FUNCTION_BLOCK FB_MqttBlindInputAdapter IMPLEMENTS I_CyclicExecution, I_MqttMessageReceiver, I_MqttDeviceDiscoveryProvider
VAR_INPUT
	POS : BYTE;	// Feedback of blind position
END_VAR
VAR_OUTPUT
	Q : BOOL;  // If new values shall be taken into blind_input. Connect this to "BLIND_INPUT.IN"
	PO : BYTE; // The position values which shall be taken into blind_input. Connect this to "BLIND_INPUT.PI"
END_VAR
VAR
	rMqttController : REFERENCE TO FB_MqttController;
	fbDeviceDiscovery : FB_MqttCoverPositionDiscovery;
	stConfig : ST_MqttCoverPositionConfiguration;
	bSetPositionOutput : BOOL; // var for cycle synchronisation
	tSendPositionUpdatesPeriod : TIME := T#1s;
	tLastPositionUpdate : TIME := T#0S;
	tCurrent : TIME;
	nLastPositionUpdateValue : BYTE;
	bStopRequested : BOOL;
END_VAR

this^.CyclicExecute();

METHOD Close : BOOL
VAR_INPUT
END_VAR
Close := this^.SetPosition(nPosition := GVL_MQTT_CONST.COVER_POSITION_CLOSED);
END_METHOD

METHOD CyclicExecute : BOOL
THIS^.tCurrent := DWORD_TO_TIME(OSCAT_BASIC.T_PLC_MS());

IF THIS^.bStopRequested THEN
	THIS^.SetPosition(nPosition := THIS^.POS);
	this^.bStopRequested := FALSE;
END_IF

THIS^.Q := THIS^.bSetPositionOutput;
THIS^.bSetPositionOutput := FALSE;

IF THIS^.tCurrent - THIS^.tLastPositionUpdate > THIS^.tSendPositionUpdatesPeriod THEN
	IF THIS^.nLastPositionUpdateValue <> THIS^.POS THEN
		THIS^.SendCurrentPosition();
		THIS^.tLastPositionUpdate := THIS^.tCurrent;
	END_IF
END_IF
END_METHOD

METHOD FB_init : BOOL
VAR_INPUT
	bInitRetains : BOOL; // if TRUE, the retain variables are initialized (warm start / cold start)
	bInCopyCode : BOOL;  // if TRUE, the instance afterwards gets moved into the copy code (online change)
	rMqttController : REFERENCE TO FB_MqttController;
	sMainTopic : STRING(255);
	sIdentifier : STRING(20);
	sName : STRING(30);
END_VAR
VAR
	stDevinfo : ST_MqttDeviceInformation;
	sTemp : STRING(255);
END_VAR
THIS^.rMqttController REF= rMqttController;

THIS^.fbDeviceDiscovery.SetMqttClient(rMqttClient := rMqttController.MqttClient);
THIS^.fbDeviceDiscovery.NodeId := GVL_MQTT_CONST.DEV_DISCOVER_NODEID;
THIS^.fbDeviceDiscovery.ObjectId := sIdentifier;

stDevinfo.identifiers := sIdentifier;
stDevinfo.manufacturer := GVL_MQTT_CONST.DEV_DISCOVER_MANUFACTURER;
stDevinfo.model := 'FB_MqttBlindInputAdapter';
stDevinfo.sw_version := GVL_CONST.SW_VERSION;
stDevinfo.name := sName;
THIS^.fbDeviceDiscovery.DeviceInformation := stDevinfo;

THIS^.stConfig.name := sName;
THIS^.stConfig.device_class := GVL_MQTT_CONST.COVER_DEV_CLASS_BLIND;
THIS^.stConfig.optimistic := FALSE;
THIS^.stConfig.unique_id := sIdentifier;
sTemp := CONCAT(STR1 := sMainTopic, STR2 := '/');
THIS^.stConfig.command_topic := CONCAT(STR1 := sTemp, STR2 := GVL_MQTT_CONST.TOPIC_COMMAND);
THIS^.stConfig.position_topic := CONCAT(STR1 := sTemp, STR2 := GVL_MQTT_CONST.TOPIC_POSITION);
THIS^.stConfig.set_position_topic := CONCAT(STR1 := sTemp, STR2 := GVL_MQTT_CONST.TOPIC_SET_POSITION);
THIS^.stConfig.payload_close := GVL_MQTT_CONST.PL_COVER_COMMAND_CLOSE;
THIS^.stConfig.payload_open := GVL_MQTT_CONST.PL_COVER_COMMAND_OPEN;
THIS^.stConfig.payload_stop := GVL_MQTT_CONST.PL_COVER_COMMAND_STOP;
THIS^.stConfig.position_closed := GVL_MQTT_CONST.COVER_POSITION_CLOSED;
THIS^.stConfig.position_open := GVL_MQTT_CONST.COVER_POSITION_OPEN;
THIS^.fbDeviceDiscovery.Configuration := THIS^.stConfig;

THIS^.rMqttController.RegisterMqttMessageReceive(
	iMqttMessageReceiver := THIS^,
	sTopic := THIS^.stConfig.command_topic);
THIS^.rMqttController.RegisterMqttMessageReceive(
	iMqttMessageReceiver := THIS^,
	sTopic := THIS^.stConfig.set_position_topic);
END_METHOD

METHOD GetMqttDeviceDiscovery : I_MqttDeviceDiscovery
GetMqttDeviceDiscovery := this^.fbDeviceDiscovery;
END_METHOD

METHOD OnMqttMessage : BOOL
VAR_INPUT
	rMqttMessage	: REFERENCE TO Tc3_IotBase.FB_IotMqttMessage;
END_VAR
VAR
	sPayload : STRING(10);
	nNewPosition : BYTE;
	bSuccess : BOOL := FALSE;
END_VAR
IF (__ISVALIDREF(rMqttMessage)) THEN
	IF rMqttMessage.CompareTopic(sTopic := THIS^.stConfig.command_topic) THEN
		IF rMqttMessage.GetPayload(pPayload := ADR(sPayload),
				nPayloadSize := 10,
				bSetNullTermination := TRUE) THEN
			IF F_StrCmp(pStr1 := ADR(sPayload), pStr2 := ADR(THIS^.stConfig.payload_close)) THEN
				THIS^.Close();
				bSuccess := TRUE;
			ELSIF F_StrCmp(pStr1 := ADR(sPayload), pStr2 := ADR(THIS^.stConfig.payload_open)) THEN
				THIS^.Open();
				bSuccess := TRUE;
			ELSIF F_StrCmp(pStr1 := ADR(sPayload), pStr2 := ADR(THIS^.stConfig.payload_stop)) THEN
				THIS^.Stop();
				bSuccess := TRUE;
			END_IF
		END_IF
	ELSIF rMqttMessage.CompareTopic(sTopic := THIS^.stConfig.set_position_topic) THEN
		IF rMqttMessage.GetPayload(pPayload := ADR(sPayload),
				nPayloadSize := 10,
				bSetNullTermination := TRUE) THEN
			nNewPosition := OSCAT_BASIC.DEC_TO_BYTE(DEC := sPayload);
			bSuccess := THIS^.SetPosition(nPosition := nNewPosition);
		END_IF
	END_IF
END_IF

OnMqttMessage := bSuccess;
END_METHOD

METHOD Open : BOOL
VAR_INPUT
END_VAR
Open := this^.SetPosition(nPosition := GVL_MQTT_CONST.COVER_POSITION_OPEN);
END_METHOD

METHOD PRIVATE SendCurrentPosition : BOOL
VAR_INPUT
END_VAR
VAR
	nPositionValue : BYTE;
	sPosValue : STRING(4);
END_VAR
IF (__ISVALIDREF(rMqttController) AND __ISVALIDREF(rMqttController.MqttClient)) THEN
	IF (rMqttController.MqttClient.bConnected) THEN
		nPositionValue := THIS^.POS;
		sPosValue := BYTE_TO_DECSTR(in := nPositionValue, iPrecision := 1);
		SendCurrentPosition := rMqttController.MqttClient.Publish(sTopic:= THIS^.stConfig.position_topic, 
			pPayload:= ADR(sPosValue), nPayloadSize:= LEN2(ADR(sPosValue)),
			eQoS:= TcIotMqttQos.AtMostOnceDelivery, bRetain:= TRUE,
			bQueue:= FALSE);
		IF SendCurrentPosition THEN
			THIS^.nLastPositionUpdateValue := nPositionValue;
		END_IF
	END_IF
END_IF
END_METHOD

METHOD SetPosition : BOOL
VAR_INPUT
	nPosition : BYTE;
END_VAR
THIS^.PO := nPosition;
THIS^.bSetPositionOutput := TRUE;
SetPosition := TRUE;
END_METHOD

METHOD Stop : BOOL
VAR_INPUT
END_VAR
THIS^.bStopRequested := TRUE;
Stop := TRUE;
END_METHOD

END_FUNCTION_BLOCK

(* stored: Version 1.1.0.1, ProductVersion 3.1.4024.5
   POU FB_MqttBlindInputAdapter: Id {cc90ac40-4d84-4ed4-9c02-9801fa611b74}, SpecialFunc None
   Method Close: Id {cc6d0557-b629-4107-b362-6c2dd8863fba}
   Method CyclicExecute: Id {73b3828a-b629-48f4-9d96-71fbc1d3121f}
   Method FB_init: Id {7246333c-b820-4b76-9a8e-f893cea0dd95}
   Method GetMqttDeviceDiscovery: Id {19a5b0fa-2797-4da3-badb-7ff858953d6d}
   Method OnMqttMessage: Id {54017421-8044-4cda-8757-be5692466d5a}
   Method Open: Id {0ab06868-9c44-46c6-92ef-0d193062c329}
   Method SendCurrentPosition: Id {53e02ceb-f931-4efe-befd-d664c589c2b7}
   Method SetPosition: Id {fe0787c0-6824-4850-a526-3e5bb2eaf9e4}
   Method Stop: Id {fd70e836-b4ab-43ca-ae50-4d70e4c3913f} *)
